{attribute addProperty BoxType "EP3314-0002-0016"}
{attribute addProperty Id "TC_TCInputs_ChannelAT %I*ARRAY[0..6] OF TC_TCInputs_Channel_4364CDB6296370WcStateAT %I*WcState_98A4DF7520.250InfoDataAT %I*InfoData_BC63D37F80100"}
{attribute addProperty CRC "3655977419"}
{attribute addProperty SizeInBites "378"}
{attribute addProperty SizeInBytes "47.25"}
TYPE EP3314_3064F862 :
STRUCT
	{attribute addProperty Name "TC_TCInputs_Channel"}
	TC_TCInputs_Channel : ARRAY[0..6] OF TC_TCInputs_Channel_4364CDB6;
	{attribute addProperty Name "WcState"}
	WcState : WcState_98A4DF75;
	{attribute addProperty Name "InfoData"}
	InfoData : InfoData_BC63D37F;
END_STRUCT
END_TYPE

(* stored: Version 1.2.0.0, ProductVersion 3.1.4024.9
   DUT EP3314_3064F862: Id {ca008a16-621e-46c6-8157-4a42f3965160} *)
